// TIA Portal V15.1 export
// export: Created 2024-05-17T05:38:43.7170449Z, ExportSetting WithDefaults, DisplayName Totally Integrated Automation Portal, DisplayVersion V15.1 Update 5, DisplayName TIA Portal Openness, DisplayVersion V15.1 Update 5, DisplayName SINAMICS Startdrive Advanced, DisplayVersion V15.1, DisplayName G130, G150, S120, S150, SINAMICS MV, S210, DisplayVersion V15.1, DisplayName G110M, G120, G120C, G120D, G120P, DisplayVersion V15.1, DisplayName STEP 7 Professional, DisplayVersion V15.1 Update 5, DisplayName STEP 7 Safety, DisplayVersion V15.1, DisplayName WinCC Professional, DisplayVersion V15.1 Update 5, DisplayName SIMATIC Visualization Architect, DisplayVersion V15.1
FUNCTION "LGBRdWrPipe" : Void   // FC6605, SCL
{ S7_Optimized_Access := 'TRUE' }
VERSION : 0.1
// stored: AutoNumber false, IsIECCheckEnabled false, SetENOAutomatically False, UDAEnableTagReadback false
   VAR_INPUT
      I_Index : Int;
      I_EnableWrite : Bool;
      I_EnableRead : Bool;
   END_VAR
   VAR_IN_OUT
      IO_Done : Bool;
      IO_Pipe : Array[1..50] of "TCPipe";
      IO_PipeData : "TCPipe";
   END_VAR
   VAR_TEMP
      RetVal : Int;
   END_VAR
BEGIN
   //------------------------------------------------------------------------------------------------
   //Handles the  writing of the data to the recipe 
   //------------------------------------------------------------------------------------------------

   //------------------------------------------------------------------------------------------------
   //Check change of input indexes and if true >>> write data to 
   //------------------------------------------------------------------------------------------------
   IF #I_EnableWrite = true THEN

       #IO_PipeData := #IO_Pipe[#I_Index];
       #IO_Done := true;

   END_IF;

   IF #I_EnableRead = true AND #IO_PipeData.PipeStart = #I_Index THEN
       #IO_Pipe[#I_Index] := #IO_PipeData;
       #IO_Done := true;

   END_IF;
END_FUNCTION
